(* IEC 61131-3 sources: InfiniteStateMachine/extracted_st/project/infinitestatemachine/function_blocks/statemachine, 3 files *)

(* ---- enter-Enter.st ---- *)
(* --- Interface --- *)
METHOD PROTECTED Enter
VAR_IN_OUT
	itfState : IState;
END_VAR

(* --- Implementation --- *)
IF Push(itfState) THEN
	itfState.Enter(THIS^);
END_IF

(* ---- goto-GoTo.st ---- *)
(* --- Interface --- *)
METHOD PUBLIC GoTo
VAR
	itfState : IState;
	fbStateMachine : StateMachine;
	iDepth : INT := 0;
END_VAR

(* --- Implementation --- *)
fbStateMachine.Jump(itfState);
WHILE iDepth < Depth() AND iDepth < fbStateMachine.Depth() AND IsSameState(AtLevel(iDepth), fbStateMachine.AtLevel(iDepth)) DO
	iDepth := iDepth + 1;
END_WHILE
WHILE Depth() > iDepth DO
	Leave();
END_WHILE
WHILE fbStateMachine.Depth() > iDepth DO
	Enter(fbStateMachine.AtLevel(iDepth));
	iDepth := iDepth + 1;
END_WHILE

(* ---- jump-Jump.st ---- *)
(* --- Interface --- *)
METHOD Jump
VAR_INPUT
	itfState : IState;
END_VAR

(* --- Implementation --- *)
iDepth := DepthOfState(itfState, ISM.gc_iMaxDepth, itfStates);
